// TwinCAT 3 PLC project Parameters
// Title: Parameters
// Company: _
// Author: Krystian Lis et al.
// ProjectVersion: 1.0.0
// Description: No more VAR PERSITANT
// ProgramVersion: 3.1.4026.9
// libraries:
//   Strings, * (_)
// project tree:
//   Persistant/ BOOL_Param.TcPOU, REAL_Param.TcPOU, DINT_Param.TcPOU, LREAL_Param.TcPOU, STR_Param.TcPOU, TIME_Param.TcPOU, UDINT_Param.TcPOU
// (motion and I/O tree: see PLC project broadcast)
// real-time tasks:
//   TASK PlcTask: cycle T#10ms, priority 20, ADS port 350
//   TASK VISU_TASK: cycle T#200000us, priority 30, ADS port 351

// ---- Persistant/BOOL_Param.TcPOU
FUNCTION_BLOCK BOOL_Param
VAR_INPUT PERSISTENT
	val				: BOOL;
END_VAR

END_FUNCTION_BLOCK

// ---- Persistant/REAL_Param.TcPOU
FUNCTION_BLOCK REAL_Param
VAR_INPUT PERSISTENT
	val			: REAL;
END_VAR

END_FUNCTION_BLOCK

// ---- Persistant/DINT_Param.TcPOU
FUNCTION_BLOCK DINT_Param
VAR_INPUT PERSISTENT
	val			: DINT;
END_VAR

END_FUNCTION_BLOCK

// ---- Persistant/LREAL_Param.TcPOU
FUNCTION_BLOCK LREAL_Param
VAR_INPUT PERSISTENT
	val			: LREAL;
END_VAR

END_FUNCTION_BLOCK

// ---- Persistant/STR_Param.TcPOU
FUNCTION_BLOCK STR_Param
VAR_INPUT PERSISTENT
	val			: Strings.Str;
END_VAR

END_FUNCTION_BLOCK

// ---- Persistant/TIME_Param.TcPOU
FUNCTION_BLOCK TIME_Param
VAR_INPUT PERSISTENT
	val			: TIME;
END_VAR

END_FUNCTION_BLOCK

// ---- Persistant/UDINT_Param.TcPOU
FUNCTION_BLOCK UDINT_Param
VAR_INPUT PERSISTENT
	val			: UDINT;
END_VAR

END_FUNCTION_BLOCK
